Fanuc KAREL source: ko00058.KL

-- PROVISIONAL review KL for V1013-1; original PC SHA256 489805f8111c15042da091ce88dc725f657e6ce86d3f48ba85356a821ef7075b
-- Incomplete behavior may be omitted. Consult companion uncertainty JSON. Do not deploy.
PROGRAM KO00058
%NOLOCKGROUP
BEGIN
  -- UNRESOLVED_PC offsets 5-12; opcodes 9D,23
  -- UNRESOLVED_PC offsets 17-69; opcodes 27,27,49,7E,AD,27,49,7E,AD,22,31,7E,4A
  -- UNRESOLVED_PC offsets 74-78; opcodes 7F
END KO00058
